PROGRAM MAIN
VAR
	PackMLTime : ARRAY[0..6] OF DINT;
	bTest: BOOL;
	bTest2: BOOL;
	result: ULINT;
END_VAR

IF bTest THEN
	PackMLTime := ULINT_TO_PackMLTime(F_GetSystemTime());
END_IF

IF bTest2 THEN
	result := PakcML_TO_TIME(PackMLTime :=PackMLTime );
END_IF

END_PROGRAM

(* stored: Version 1.1.0.1, ProductVersion 3.1.4024.11
   POU MAIN: Id {fd831da4-b786-496f-a354-4672dd96d1fd}, SpecialFunc None *)
